{attribute 'qualified_only'}
VAR_GLOBAL
	bStartPB : BOOL;
	bStopPB : BOOL;
	
	bStartTB : BOOL;
	bStopTB : BOOL;
	
	bIndicator1 : BOOL;
	bIndicator2 : BOOL;
	
	
	btn : BOOL;
	dayNightSwitch : BOOL;
		
	led1_1 : BOOL;
	led2_1 : BOOL;
	led2_2 : BOOL;
	led3 : BOOL;
	led4_1 : BOOL;
	led4_2 : BOOL;
	led4_3 : BOOL;
	//led4_4 : BOOL;
	
	
END_VAR

(* stored: Version 1.1.0.1, ProductVersion 3.1.4024.12
   GVL HMI: Id {75a31c87-ad94-45c2-bd29-497ae1135acc} *)
